(* Schneider Machine Expert - Basic project ReglageHoraire, file version 1.2.0.0 *)

HARDWARE
  Cpu 0: TM221ME16T/G
  EthernetConfiguration: NetworkName=M221, IpAllocationMode=FixedAddress, IpAddress=0.0.0.0, SubnetMask=0.0.0.0
  SerialLineConfiguration: Baud=Baud19200, Parity=ParityEven, DataBits=DataBits8, StopBits=StopBits1, PhysicalMedium=PhysicalMediumRs485, TransmissionMode=TransmissionModeModbusRtu, SlaveId=1, Addressing=SlaveAddressing
  MastTask: UsePeriodScanMode=false, PeriodScan=100
  FastTask: Period=255
  CpuBehavior: StartingMode=StartInRun, AutoSaveRamOnEeprom=true, WatchdogPeriod=250

SYMBOLS  (address, symbol, comment, settings)
  %S50      SB_RTCUPDATE  "Set to 1, this bit allows to update the date and time"
  %SW49     SW_RTCDAY  "RTC Function: contains in BCD xN Day of the week (N=1 for Monday)"
  %SW50     SW_RTCSEC  "RTC Function: contains in BCD 00SS Seconds"
  %SW51     SW_RTCHHMM  "RTC Function: contains in BCD HHMM: hour and minute"
  %SW52     SW_RTCMMDD  "RTC Function: contains in BCD MMDD: month and day"
  %SW53     SW_RTCCCYY  "RTC Function: contains in BCD CCYY: century and year"

POU Nouveau POU
  (* SectionNumber=1, IsGrafcet=false *)

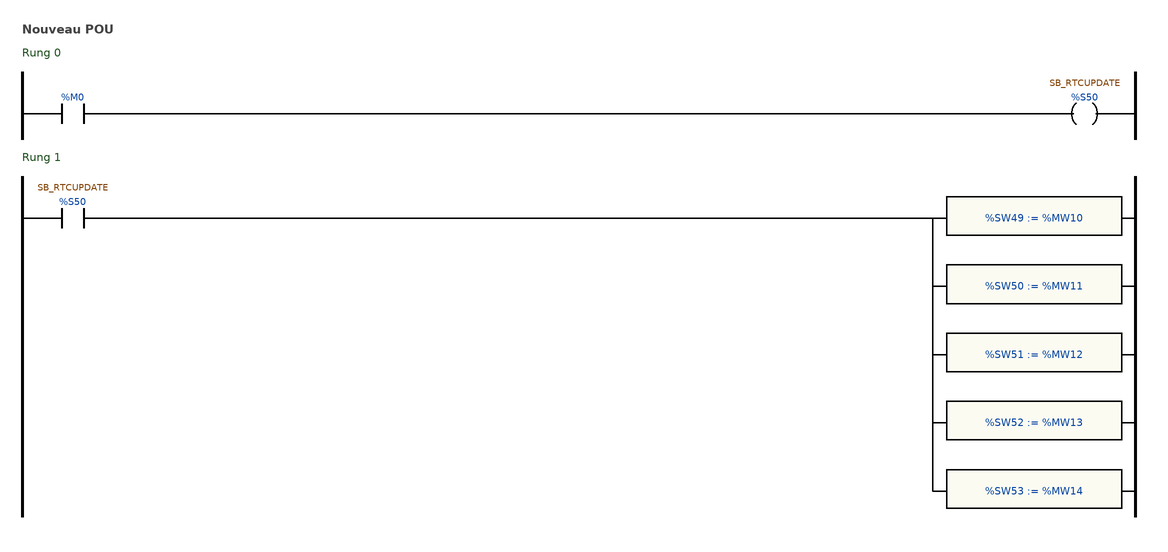

// Rung 0
  LD %M0
  ST %S50                 (* SB_RTCUPDATE *)
  // as ST:
  //   SB_RTCUPDATE := %M0;

// Rung 1
  LD %S50                 (* SB_RTCUPDATE *)
  [%SW49 := %MW10]        (* SW_RTCDAY *)
  [%SW50 := %MW11]        (* SW_RTCSEC *)
  [%SW51 := %MW12]        (* SW_RTCHHMM *)
  [%SW52 := %MW13]        (* SW_RTCMMDD *)
  [%SW53 := %MW14]        (* SW_RTCCCYY *)
  // as ST:
  //   IF SB_RTCUPDATE THEN SW_RTCDAY := %MW10; END_IF;
  //   IF SB_RTCUPDATE THEN SW_RTCSEC := %MW11; END_IF;
  //   IF SB_RTCUPDATE THEN SW_RTCHHMM := %MW12; END_IF;
  //   IF SB_RTCUPDATE THEN SW_RTCMMDD := %MW13; END_IF;
  //   IF SB_RTCUPDATE THEN SW_RTCCCYY := %MW14; END_IF;
